Staubli VAL3: usrSelect.pgx

public program usrSelect(num& nWhichBttn (dimensions=1))
begin
  nWhichBttn=-1
  do
    nWhichBttn=(get()-270)
  until ((nWhichBttn==1) or (nWhichBttn==8))
end
